PROGRAM P_Demo_F_BA_DiffPtr
VAR
    argPAddr1                      : PVOID                          := 0; // pAddr1
    argPAddr2                      : PVOID                          := 0; // pAddr2
    fnReturn                       : UDINT; // 返回值
END_VAR

// =============================================================================
// Tc3_BA2_Common.F_BA_DiffPtr 演示程序
// =============================================================================
// 场景：在大缓冲区里找到某个标志位的位置后，反算出该位置距离缓冲区起始的偏移。
//
// 价值：跨 x86/x64 平台自动正确；手写 `pAddr1 - pAddr2` 在 x64 上会截断造成偏移错误。
//
// 验证：登录 PLC 后，按例程内变量在线写值；监视输出 / 返回值，结合 §1 功能
//       简述的预期行为对照（详见配套 .md 文档 §7 业务场景）。
//
// 验证步骤：
//   1. 右键 PLC 项目下 POUs 文件夹 → Add → Existing Item → 选本 .TcPOU 文件
//   2. 引用 Tc3_BA2_Common（References → Add library）
//   3. 编译 → 登录 → 运行；按上方『验证』指引在线写值观察
// =============================================================================

fnReturn := F_BA_DiffPtr(
    pAddr1                   := argPAddr1,
    pAddr2                   := argPAddr2
);

END_PROGRAM

(* stored: Version 1.1.0.1, ProductVersion 3.1.4024.5
   POU P_Demo_F_BA_DiffPtr: Id {01cb3aa4-f055-551e-8f2f-e85b1f52670e}, SpecialFunc None *)
